// Provide logging 
FUNCTION_BLOCK FB_TcLogger IMPLEMENTS I_Logger, I_LogLevel
VAR_INPUT
	eLogLevel:				E_LogLevel:= E_LogLevel.Info;
END_VAR
VAR
	fbSourceInfo:			FB_TcSourceInfo;
	aAlarm:					ARRAY[0..99] OF FB_TcAlarm; 	// Message store
    nAlarm:					UINT;                     		// Message count
	bAlarm:					ARRAY[0..99] OF BOOL; 	// Message store
	{attribute 'hide'} 
	nIndex: 				UINT;
	{attribute 'hide'} 
	nTimestamp:				LINT;
END_VAR

// https://peterzerlauth.com/

// @ToDo

// nIndex := 0;
// WHILE nIndex < nAlarm DO
//     IF bAlarm[nIndex] = TRUE THEN
// 		bAlarm[nIndex]:= FALSE;
//     END_IF
//     nIndex := nIndex + 1;
// END_WHILE
// M_Reset:= TRUE;
// // https://peterzerlauth.com/
// 
// IF nTimestamp < TwinCAT_SystemInfoVarList._TaskInfo[GETCURTASKINDEXEX()].DcTaskTime THEN // 1 second = 1e9 ns
// 	nTimestamp := TwinCAT_SystemInfoVarList._TaskInfo[GETCURTASKINDEXEX()].DcTaskTime + 1000000000;
// 	nIndex:= 0;
// 	WHILE nIndex < nAlarm DO
// 		IF bAlarm[nIndex] THEN
// 			IF aAlarm[nIndex].eSeverity <= LogLevel_To_TcEventSeverity(E_LogLevel.Warning) THEN
// 				bAlarm[nIndex]:= FALSE;
// 			END_IF
// 			nIndex := nIndex + 1;
// 		ELSE
// 			aAlarm[nIndex].Release
// 			nMessages := nMessages - 1;
// 			RETURN;
// 		END_IF
// 	END_WHILE
// END_IF

METHOD PUBLIC M_Log : BOOL
VAR_INPUT
	fbMessage:			FB_Message;
END_VAR
VAR
	sArgument:			STRING;
	nPosition: 			INT;
END_VAR
IF eLogLevel > fbMessage.eLogLevel THEN
	M_Log:= TRUE;
	RETURN;
END_IF

IF nAlarm > 99 THEN 
	RETURN;
END_IF

// Skip if same sMessage already exists
nIndex := 0;
WHILE nIndex < nAlarm DO
    IF aAlarm[nIndex].EqualsToEventEntry(TC_EVENT_CLASSES.Tc3_Event, fbMessage.nID, LogLevel_To_TcEventSeverity(fbMessage.eLogLevel))  THEN
		bAlarm[nIndex]:= TRUE;
        M_Log := TRUE;
        RETURN;
    END_IF
    nIndex := nIndex + 1;
END_WHILE

// prepare
fbSourceInfo.Clear();
fbSourceInfo.sName:= fbMessage.sSource;
aAlarm[nAlarm].Create(TC_EVENT_CLASSES.Tc3_Event,  fbMessage.nID, LogLevel_To_TcEventSeverity(fbMessage.eLogLevel), FALSE, fbSourceInfo);
aAlarm[nAlarm].ipArguments.Clear();

// Split and add arguments
nPosition := FIND('$R', fbMessage.sArguments);
WHILE nPosition > 0 DO
    sArgument := LEFT(fbMessage.sArguments, nPosition - 1);
    aAlarm[nAlarm].ipArguments.AddString(sArgument);
    fbMessage.sArguments:= RIGHT(fbMessage.sArguments, LEN(fbMessage.sArguments) - (nPosition + 1));
    nPosition := FIND('$R', fbMessage.sArguments);
END_WHILE;

// Raise alarm
aAlarm[nAlarm].Raise(fbMessage.nTimestamp);

nAlarm := nAlarm + 1;
M_Log := TRUE;
END_METHOD

METHOD M_Reset : BOOL
VAR_INPUT
END_VAR
nIndex := 0;
WHILE nIndex < nAlarm DO
    IF bAlarm[nIndex] = TRUE THEN
		bAlarm[nIndex]:= FALSE;
    END_IF
    nIndex := nIndex + 1;
END_WHILE
M_Reset:= TRUE;
END_METHOD

{attribute 'OPC.UA.DA.Property' := '1'}
{attribute 'monitoring' := 'variable'}
PROPERTY PUBLIC P_LogLevel : E_LogLevel
GET
P_LogLevel:= eLogLevel;
END_GET
SET
eLogLevel:= P_LogLevel;
END_SET
END_PROPERTY

END_FUNCTION_BLOCK

(* stored: Version 1.1.0.1
   POU FB_TcLogger: Id {c4bb1a5e-d8ae-49cb-90d9-702eaf5363d5}, SpecialFunc None
   Method M_Log: Id {6fe90735-819e-4754-991c-316c9aee4d7c}
   Method M_Reset: Id {49b80e31-c5f7-4f9f-b087-49844ffe0726}
   Property P_LogLevel: Id {f86a40a0-98fd-40f4-a32f-52729e621278}
   Get Get: Id {65712a2e-9ca7-492d-83fc-203b71a5ffed}
   Set Set: Id {a818a2a2-1395-45f7-a05b-b64f5da416d8} *)
